FUNCTION AxesAlphaUnitsToDeg : LREAL
VAR_INPUT
    units : AxesAlphaUnits;
    value : LREAL;
END_VAR
VAR
END_VAR

CASE units OF
    AxesAlphaUnits.RADIANS:
        AxesAlphaUnitsToDeg := RAD_TO_DEG(value);
    AxesAlphaUnits.DEGREES:
        AxesAlphaUnitsToDeg := value; 
    AxesAlphaUnits.HOURS:
        AxesAlphaUnitsToDeg := HOUR_TO_DEG(value);   
END_CASE

END_FUNCTION

(* stored: Version 1.1.0.1, ProductVersion 3.1.4019.2
   POU AxesAlphaUnitsToDeg: Id {b3b3add3-a4aa-44bb-884f-9933fbc8bfdc}, SpecialFunc None *)
